(*			
	RAFALOS
	Rafał Osajda		23.09.2025		TC 4024.66
	Struktura pomocnicza potrzeba do wiazania zmiennych
*)
TYPE ST_BaseControlElement_HMI_Link :
STRUCT
	stBaseLoggerElement				: ST_BaseLoggerElement_HMI;
	stBaseComponent					: ST_BaseComponent_HMI;
	stBaseControlElement			: ST_BaseControlElement_HMI;
END_STRUCT
END_TYPE

(* stored: Version 1.1.0.1
   DUT ST_BaseControlElement_HMI_Link: Id {50dc1360-1024-0da2-163a-cf7aa292fa73} *)
